Staubli VAL3: getPath.pgx

program getPath(string& x_sType[] (dimensions=1))
  local num l_nPos
  local string l_sPath
  local num i
begin
  // get the TypePath
  call saveData:getPathInstr(x_sType,x_sType)
end
